FUNCTION_BLOCK FB_GovernorTest

VAR
	istep			:		UINT;
	bStart			:		BOOL;

	fbGovernor	:	FB_GovernorSerialCom;
END_VAR

CASE istep OF
	0: //Trigger
		IF bStart THEN
			bStart := FALSE;
			istep := 10;
		END_IF
		
	10: //Init		
		fbGovernor.Init();
		fbGovernor.Timeout := 1000;
		fbGovernor.ScanTime := 1;
		istep := 20;
		
	20: //Running
		IF fbGovernor.Run() THEN
			istep := 30;
		END_IF
		
	30: //Stopped
		
END_CASE

fbGovernor();

END_FUNCTION_BLOCK

(* stored: Version 1.1.0.1, ProductVersion 3.1.4024.12
   POU FB_GovernorTest: Id {caeeb0d8-549a-4820-8104-7f654818a633}, SpecialFunc None *)
